// TIA Portal V18 export
// export: Created 2025-12-01T17:51:28.8249822Z, ExportSetting None, DisplayName Totally Integrated Automation Portal, DisplayVersion V18 Update 5, DisplayName TIA Portal Openness, DisplayVersion V18 Update 5, DisplayName TIA Portal Teamcenter Gateway, DisplayVersion V18, DisplayName TIA Portal Version Control Interface, DisplayVersion V18, DisplayName STEP 7 Professional, DisplayVersion V18 Update 5, DisplayName STEP 7 Safety, DisplayVersion V18, DisplayName WinCC Professional, DisplayVersion V18 Update 5
DATA_BLOCK "Station8LoadData"   // DB524
{ S7_Optimized_Access := 'FALSE' }
// stored: AutoNumber false
   VAR
      "PLC.PartTypeID" : Int;
      "PLC.Station8RecipeNo" : Int;
      "PLC.Station8DMXCode" : String[128];
      Spare : Byte;
      "MES.ErrorCode" : Int;
      "MES.StatusBits" : DInt;
      "MES.Cycle_ID" : DInt;
      "MES.Unit_ParttypeID" : Int;
   END_VAR
BEGIN
END_DATA_BLOCK
